(* PLC project Untitled1, Beckhoff Automation GmbH TF6420 Database Server Query Analyser 1.0.0.0 *)
(* stored: creationDateTime 2021-07-19T09:40:43, modificationDateTime 2021-07-19T09:40:43 *)

TYPE ST_SelectStruct : STRUCT
  _name : STRING(255);
  _dint : DINT;
  _real : REAL;
  _lreal : LREAL;
  _date : ARRAY[0..255] OF BYTE;
END_STRUCT;
END_TYPE
